// TIA Portal V16.AddIn export
// export: Created 2019-07-15T20:10:39.7344093Z, ExportSetting WithDefaults, DisplayName Totally Integrated Automation Portal, DisplayVersion V16, DisplayName TIA Portal Version Control Interface, DisplayVersion V16, DisplayName TIA Portal Openness, DisplayVersion V16, DisplayName Feature Cycle 3 TIA Portal, DisplayVersion V16, DisplayName STEP 7 Professional, DisplayVersion V16, DisplayName STEP 7 Safety, DisplayVersion V16, DisplayName WinCC Professional, DisplayVersion V16
TYPE "typeProductCounter"
// stored: IsFailsafeCompliant false
   STRUCT
      trigger : Bool;   // Trigger
      reset : Bool;   // Resetting of total product counter
      count : DInt;   // Counter of total products (resettable)
      accCount : DInt;   // Accumulated counter of total products (non resettable)
   END_STRUCT;
END_TYPE
